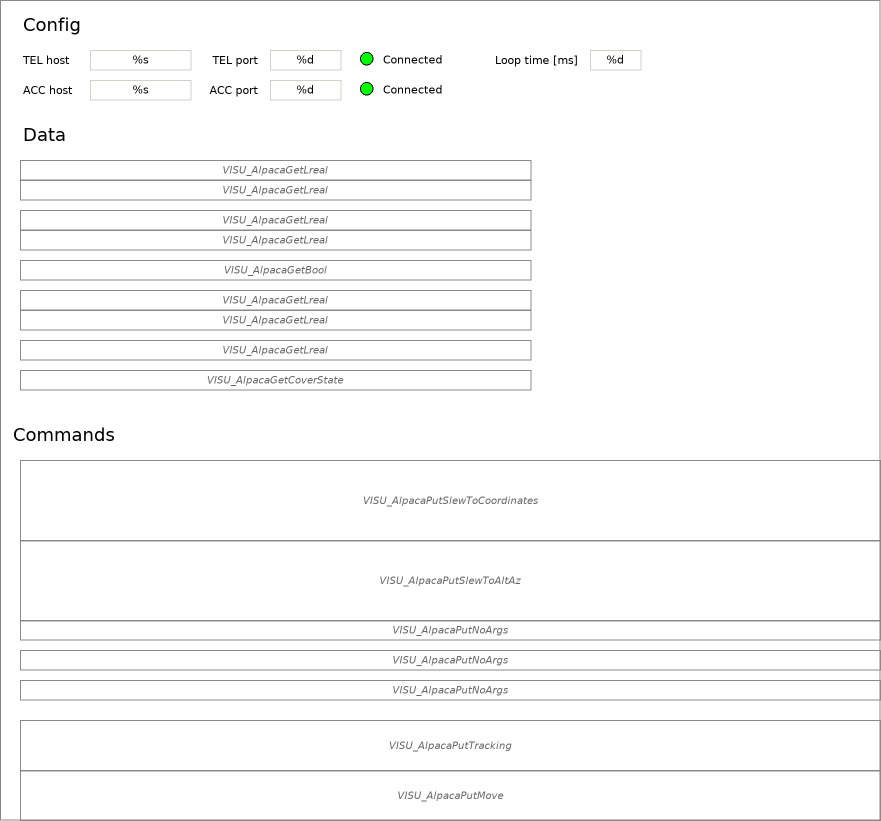
VISUALIZATION VISU_AsaTelescope  // 881x821
VAR_IN_OUT
	fbInstance : FB_AsaTelescope;
END_VAR
    Frame (20,160 511x20)
        shows VISU_AlpacaGetLreal(stInstance := fbInstance.stData.stRightAscension)
    Frame (20,180 511x20)
        shows VISU_AlpacaGetLreal(stInstance := fbInstance.stData.stDeclination)
    Frame (20,210 511x20)
        shows VISU_AlpacaGetLreal(stInstance := fbInstance.stData.stAzimuth)
    Frame (20,230 511x20)
        shows VISU_AlpacaGetLreal(stInstance := fbInstance.stData.stAltitude)
    Frame (20,290 511x20)
        shows VISU_AlpacaGetLreal(stInstance := fbInstance.stData.stTargetRightAscension)
    Frame (20,310 511x20)
        shows VISU_AlpacaGetLreal(stInstance := fbInstance.stData.stTargetDeclination)
    Frame (20,260 511x20)
        shows VISU_AlpacaGetBool(stInstance := fbInstance.stData.stSlewing)
    Label (20,120 150x30), "Data"
    Label (10,420 211x30), "Commands"
    Frame (20,460 861x81)
        shows VISU_AlpacaPutSlewToCoordinates(stInstance := fbInstance.stCommands.stSlewToCoo)
    Frame (20,540 861x81)
        shows VISU_AlpacaPutSlewToAltAz(stInstance := fbInstance.stCommands.stSlewToAltAz)
    Frame (20,650 861x20)
        shows VISU_AlpacaPutNoArgs(stInstance := fbInstance.stCommands.stOpenCover)
    Frame (20,680 861x20)
        shows VISU_AlpacaPutNoArgs(stInstance := fbInstance.stCommands.stCloseCover)
    Frame (20,720 861x51)
        shows VISU_AlpacaPutTracking(stInstance := fbInstance.stCommands.stTracking)
    Frame (20,340 511x20)
        shows VISU_AlpacaGetLreal(stInstance := fbInstance.stData.stM2Position)
    Frame (20,770 861x51)
        shows VISU_AlpacaPutMove(stInstance := fbInstance.stCommands.stM2Move)
    Frame (20,370 511x20)
        shows VISU_AlpacaGetCoverState(stInstance := fbInstance.stData.stCoverState)
    Frame (20,620 861x20)
        shows VISU_AlpacaPutNoArgs(stInstance := fbInstance.stCommands.stAbortSlew)
    Label (20,10 150x30), "Config"
    Label (20,50 71x21), "TEL host"
    Textfield (90,50 101x20), "%s", text variable: fbInstance.sTelHost
        OnMouseClick: write the text variable via Default
    Textfield (270,50 71x20), "%d", text variable: fbInstance.nTelPort
        OnMouseClick: write the text variable via Default
    Label (200,50 61x21), "TEL port"
    Textfield (590,50 51x20), "%d", text variable: fbInstance.nLoopTime
        OnMouseClick: write the text variable via Default
    Label (490,50 91x21), "Loop time [ms]"
    Label (20,80 71x21), "ACC host"
    Textfield (90,80 101x20), "%s", text variable: fbInstance.sAccHost
        OnMouseClick: write the text variable via Default
    Textfield (270,80 71x20), "%d", text variable: fbInstance.nAccPort
        OnMouseClick: write the text variable via Default
    Label (200,80 61x21), "ACC port"
    Ellipse (360,52 13x13), colour toggle: NOT fbInstance.bTelConnected
    Ellipse (360,82 13x13), colour toggle: NOT fbInstance.bAccConnected
    Label (380,50 91x20), "Connected"
    Label (380,80 91x20), "Connected"
END_VISUALIZATION

(* stored: Version 1.1.0.1, ProductVersion 3.1.4024.12
   Visu VISU_AsaTelescope: Id {b9f29362-eb86-4dd8-be49-326337dec16f} *)
